// TIA Portal project "SVO_Lib" (V14)

(* hardware
DEVICE "S7300/ET200M station_1"  S7-300 station
   slot 0: "Rail_0"  Rail  6ES7 390-1***0-0AA0
   slot 2: "PLC_300"  CPU 315-2 PN/DP  6ES7 315-2EH14-0AB0  V3.2
      slot 2: "PROFINET interface_1"  PN-IO
         slot 1: "Port_1"  Port
         slot 2: "Port_2"  Port
   slot 4: "DI 8x120/230VAC_1"  DI8 x 230VAC  6ES7 321-1FF01-0AA0
DEVICE "S7-1200 station_1"  S7-1200 Station
   slot 0: "Rack_0"  S7-1200 Rack  Rack  V1.0
   slot 1: "PLC_1200"  CPU 1217C DC/DC/DC  6ES7 217-1AG40-0XB0  V4.2
DEVICE "HMI_1"  TP900 Comfort
   slot 0: "TP900 Comfort"  TP900 Comfort  6AV2 124-0JC01-0AX0  14.0.1.0
   slot 1: "HMI_RT_1"  TP900 Comfort  6AV2 124-0JC01-0AX0  14.0.1.0
   slot 5: "HMI_1.IE_CP_1"  PROFINET Interface  14.0.1.0
      slot 1: "PROFINET Interface_1"  PROFINET Interface
         slot 1: "Port_1"  Port
         slot 2: "Port_2"  Port
   slot 7: "HMI_1.MPI/DP_CP_1"  MPI/DP Interface  14.0.1.0
*)

// ===== PLC "PLC_300"  CPU 315-2 PN/DP =====

VAR_GLOBAL   // PLC tag table "Default tag table"
   "Tag_3" AT %M1.5 : Bool;
   "Tag_4" AT %M2.0 : Bool;
   "Tag_5" AT %M2.1 : Bool;
   "Tag_6" AT %M2.2 : Bool;
   "Tag_7" AT %MW4 : Int;
   "i0.0" AT %I0.0 : Bool;
   "i0.1" AT %I0.1 : Bool;
   "i0.2" AT %I0.2 : Bool;
   "i0.3" AT %I0.3 : Bool;
   "i0.4" AT %I0.4 : Bool;
   "i0.5" AT %I0.5 : Bool;
   "i0.6" AT %I0.6 : Bool;
   "i0.7" AT %I0.7 : Bool;
   "Tag_1" AT %M3.0 : Bool;
   "Tag_2" AT %M2.5 : Bool;
   "Tag_8" AT %M2.7 : Bool;
   "Tag_9" AT %M2.6 : Bool;
   "Tag_10" AT %MW20 : Int;
   "Tag_11" AT %MW22 : Int;
   "Tag_12" AT %MW24 : Int;
   "Tag_13" AT %MB26 : Byte;
   "Tag_14" AT %MB27 : Byte;
   "Tag_15" AT %MB28 : Byte;
   "Tag_16" AT %MB29 : Byte;
   "Tag_17" AT %MB30 : Byte;
   "Tag_18" AT %MB31 : Byte;
   "Tag_19" AT %MB32 : Byte;
   "Tag_20" AT %MB33 : Byte;
END_VAR

VAR_GLOBAL CONSTANT   // PLC tag table "Default tag table"
   "T" : Bool := 1;
   "T2" : Bool := true;
END_VAR

VAR_GLOBAL   // PLC tag table "PLCTagsKernel"
   "Blink0_1s" AT %M10.0 : Bool;   // Frequency 10Гц
   "Blink0_2s" AT %M10.1 : Bool;   // Frequency 5Гц
   "Blink0_4s" AT %M10.2 : Bool;   // Frequency 2,5Гц
   "Blink0_5s" AT %M10.3 : Bool;   // Frequency 2Гц
   "Blink0_8s" AT %M10.4 : Bool;   // Frequency 1,25Гц
   "Blink1_0s" AT %M10.5 : Bool;   // Frequency 1Гц
   "Blink1_6s" AT %M10.6 : Bool;   // Frequency 0,625Гц
   "Blink2_0s" AT %M10.7 : Bool;   // Frequency 0,5Гц
   "False0" AT %M0.0 : Bool;   // Always 0 [No]
   "True1" AT %M0.1 : Bool;   // Always 1 [Yes]
   "PLC_Run" AT %M0.2 : Bool;   // PLC is run. [0:Stop, 1:Run]
   "COM_RST" AT %M0.3 : Bool;   // PLC was restart. [0:Stop or Run, 1:First cycle]
   "Dummy" AT %M0.6 : Bool;   // Do nothing.
   "Temp" AT %M0.7 : Bool;   // Will be change.[Mark from programmer]
   "PLC_Runing" AT %M0.4 : Bool;
END_VAR

TYPE "udtDI"
   STRUCT
      ibInput : Bool := false;   // Input signal from DI
      ibSimulationOn : Bool := false;   // When simulation is on Out = 1 [0:Off, 1:On]
      ibSensorsBipolar : Bool := false;   // [0:Unopolar,1:Bipolar]
      ibEnUseDelay : Bool := true;   // Enable use delay [0:Disable,1:Enable]
      iiOnDelaySP : Int := 1;   // Set point on delay [s]
      iiOffDelaySP : Int := 1;   // Set point off delay [s]
      ibBlink1s : Bool := false;   // A flickering signal with a frequency of 1s.
      obOut : Bool := false;   // Output signal to user program.
      niCountDelayOn : Int := 0;   // Time passed after on. Out memory for save.
      niCountDelayOff : Int := 0;   // Time passed after off. Out memory for save.
      nwStatusWord : Word := 16#0;   // Status word.
   END_STRUCT;
END_TYPE

DATA_BLOCK "diMunitorByDI"   // DB1
{ S7_Optimized_Access := 'FALSE' }
VERSION : 0.1
// stored: InstanceOfName fMonitorByDI
"fMonitorByDI"
BEGIN
END_DATA_BLOCK

DATA_BLOCK "O"   // DB2
{ S7_Optimized_Access := 'FALSE' }
VERSION : 0.1
   VAR
      DI : Array[0..100] of "udtDI";
   END_VAR
BEGIN
END_DATA_BLOCK

DATA_BLOCK "diMunitorByDI2"   // DB3
{ S7_Optimized_Access := 'FALSE' }
VERSION : 0.1
// stored: InstanceOfName fMonitorByDI
"fMonitorByDI"
BEGIN
END_DATA_BLOCK

DATA_BLOCK "fConvertWordToBits_DB"   // DB4
{ S7_Optimized_Access := 'FALSE' }
VERSION : 0.1
// stored: InstanceOfName fConvertWordToBits
"fConvertWordToBits"
BEGIN
END_DATA_BLOCK

DATA_BLOCK "fConvertByteToBits_DB"   // DB6
{ S7_Optimized_Access := 'FALSE' }
VERSION : 0.1
// stored: InstanceOfName fConvertByteToBits
"fConvertByteToBits"
BEGIN
END_DATA_BLOCK

FUNCTION_BLOCK "fConvertWordToBits"   // FB1, SCL
{ S7_Optimized_Access := 'FALSE' }
VERSION : 0.1
   VAR_INPUT
      iWord : Word := 16#0000;
   END_VAR
   VAR_OUTPUT
      oBit00 : Bool;
      oBit01 : Bool;
      oBit02 : Bool;
      oBit03 : Bool;
      oBit04 : Bool;
      oBit05 : Bool;
      oBit06 : Bool;
      oBit07 : Bool;
      oBit08 : Bool;
      oBit09 : Bool;
      oBit10 : Bool;
      oBit11 : Bool;
      oBit12 : Bool;
      oBit13 : Bool;
      oBit14 : Bool;
      oBit15 : Bool;
   END_VAR
   VAR_TEMP
      tWord : Word;
      arrayATtWord AT tWord : Array[0..15] of Bool;
   END_VAR
BEGIN
   (*
   Autor: Svinarenko V.O.
   Version : 1.0
   Notes:
   This function can unpack input word to bool.
   *)

   #tWord := #iWord;

   #oBit00 := #arrayATtWord[8];
   #oBit01 := #arrayATtWord[9];
   #oBit02 := #arrayATtWord[10];
   #oBit03 := #arrayATtWord[11];
   #oBit04 := #arrayATtWord[12];
   #oBit05 := #arrayATtWord[13];
   #oBit06 := #arrayATtWord[14];
   #oBit07 := #arrayATtWord[15];
   #oBit08 := #arrayATtWord[0];
   #oBit09 := #arrayATtWord[1];
   #oBit10 := #arrayATtWord[2];
   #oBit11 := #arrayATtWord[3];
   #oBit12 := #arrayATtWord[4];
   #oBit13 := #arrayATtWord[5];
   #oBit14 := #arrayATtWord[6];
   #oBit15 := #arrayATtWord[7];
END_FUNCTION_BLOCK

FUNCTION_BLOCK "fConvertBitsToWord"   // FB2, SCL
{ S7_Optimized_Access := 'FALSE' }
VERSION : 0.1
   VAR_INPUT
      iBit00 : Bool := FALSE;
      iBit01 : Bool := FALSE;
      iBit02 : Bool := FALSE;
      iBit03 : Bool := FALSE;
      iBit04 : Bool := FALSE;
      iBit05 : Bool := FALSE;
      iBit06 : Bool := FALSE;
      iBit07 : Bool := FALSE;
      iBit08 : Bool := FALSE;
      iBit09 : Bool := FALSE;
      iBit10 : Bool := FALSE;
      iBit11 : Bool := FALSE;
      iBit12 : Bool := FALSE;
      iBit13 : Bool := FALSE;
      iBit14 : Bool := FALSE;
      iBit15 : Bool := FALSE;
   END_VAR
   VAR_OUTPUT
      oWord : Word;
   END_VAR
   VAR_TEMP
      tWord : Word;
      arrayTWord AT tWord : Array[0..15] of Bool;
   END_VAR
BEGIN
   (*
   Autor: Svinarenko V.O.
   Version : 1.0
   Notes:
   This function can pack input bool to word.
   *)    
   #arrayTWord[0] := #iBit08;
   #arrayTWord[1] := #iBit09;
   #arrayTWord[2] := #iBit10;
   #arrayTWord[3] := #iBit11;
   #arrayTWord[4] := #iBit12;
   #arrayTWord[5] := #iBit13;
   #arrayTWord[6] := #iBit14;
   #arrayTWord[7] := #iBit15;
   #arrayTWord[8] := #iBit00;
   #arrayTWord[9] := #iBit01;
   #arrayTWord[10] := #iBit02;
   #arrayTWord[11] := #iBit03;
   #arrayTWord[12] := #iBit04;
   #arrayTWord[13] := #iBit05;
   #arrayTWord[14] := #iBit06;
   #arrayTWord[15] := #iBit07;

   #oWord := #tWord;
END_FUNCTION_BLOCK

FUNCTION_BLOCK "fMonitorByAI"   // FB3, SCL
{ S7_Optimized_Access := 'FALSE' }
VERSION : 0.1
   VAR_INPUT
      iiSCALE_IN : Int;   // Input value from analog input (PIW).
      iiSCALE_HI_Lim : Real := 100.0;   // High limit.
      iiSCALE_LO_Lim : Real := 0.0;   // Low limit.
      irLimHH : Real := 95.0;   // High alarm limit.
      irLimH : Real := 90.0;   // High warning limit.
      irHTL : Real := 60.0;   // High tolerant limit.
      irSP : Real := 50.0;   // Set point
      irLTL : Real := 40.0;   // Low tolerant limit.
      irLimL : Real := 10.0;   // Low warning limit.
      irLimLL : Real := 5.0;   // Low alarm limit.
      ibSimulationOn : Bool;
      ibBipolar : Bool := false;   // 0:unipolar, 1:Bipolar
      ibDoUseHiLim : Bool := true;   // 0: Do not use; 1: Use.
      ibDoUseLoLim : Bool := true;   // 0: Do not use; 1: Use.
   END_VAR
BEGIN


   // "fAICheckInputParam"(irLimHH:=#irLimHH,
   //                      irLimH:=#irLimH,
   //                      irLimL:=#irLimL,
   //                      irLimLL:=#irLimLL,
   //                      obParamOk=>_bool_out_);

   // "fAIScale"(ibBipolar:=#ibBipolar,
   //            iiSCALE_IN:=#iiSCALE_IN,
   //            iiSCALE_HI_Lim:=#iiSCALE_HI_Lim,
   //            iiSCALE_LO_Lim:=#iiSCALE_LO_Lim,
   //            orPV=>_real_out_);


   // "fAICheckLim"(irPV:=_real_in_,
   //               irLimHH:=#irLimHH,
   //               irLimH:=#irLimH,
   //               irHTL:=#irHTL,
   //               irLTL:=#irLTL,
   //               irLimL:=#irLimL,
   //               irLimLL:=#irLimLL,
   //               ibDoUseHiLim:=#ibDoUseHiLim,
   //               ibDoUseLoLim:=#ibDoUseLoLim,
   //               obFlt=>_bool_out_,
   //               obWrn=>_bool_out_,
   //               obTolerant=>_bool_out_,
   //               obFltHH=>_bool_out_,
   //               obWrnH=>_bool_out_,
   //               obWrnL=>_bool_out_,
   //               obFltLL=>_bool_out_);

   (*
   Status 
   0 Bag - Red
   1 HH - Red
   2 H - Yelow
   3 N - Gray
   4 T - Green
   5 N - Gray
   6 L - Yelow
   7 LL - Red
   *)
END_FUNCTION_BLOCK

FUNCTION_BLOCK "fValve"   // FB4, SCL
{ S7_Optimized_Access := 'FALSE' }
VERSION : 0.1
   VAR_INPUT
      ibAutoMode : Bool;
      ibManMode : Bool;
      ibAutoGoOpen : Array[0..7] of Bool;
      ibManGoOpenFromHMI : Bool;
      ibManGoOpenFromBtnFlipFlop : Bool;
      ibManGoOpenFromSwich : Bool;
      ibManGoOpenFromBtnStart : Bool;
      ibManGoOpenFromBtnStop : Bool;
      ibLook : Bool;
      ibValveIsOpen : Bool;
      ibValveIsClose : Bool;
      iiTime : Int;
   END_VAR
BEGIN
END_FUNCTION_BLOCK

FUNCTION_BLOCK "fConvertByteToBits"   // FB5, SCL
{ S7_Optimized_Access := 'FALSE' }
VERSION : 0.1
   VAR_INPUT
      iByte : Byte := 16#0000;
   END_VAR
   VAR_OUTPUT
      oBit00 : Bool;
      oBit01 : Bool;
      oBit02 : Bool;
      oBit03 : Bool;
      oBit04 : Bool;
      oBit05 : Bool;
      oBit06 : Bool;
      oBit07 : Bool;
   END_VAR
   VAR_TEMP
      tByte : Byte;
      arrayATtByte AT tByte : Array[0..7] of Bool;
   END_VAR
BEGIN
   (*
   Autor: Svinarenko V.O.
   Version : 1.0
   Notes:
   This function can unpack input byte to bool.
   *)

   #tByte := #iByte;

   #oBit00 := #arrayATtByte[0];
   #oBit01 := #arrayATtByte[1];
   #oBit02 := #arrayATtByte[2];
   #oBit03 := #arrayATtByte[3];
   #oBit04 := #arrayATtByte[4];
   #oBit05 := #arrayATtByte[5];
   #oBit06 := #arrayATtByte[6];
   #oBit07 := #arrayATtByte[7];
END_FUNCTION_BLOCK

FUNCTION_BLOCK "fMonitorByDI"   // FB50, SCL
TITLE = fMunitorByDI
{ S7_Optimized_Access := 'FALSE' }
AUTHOR : SVO
FAMILY : Munitor
VERSION : 1.2
   VAR_INPUT
      ibInput : Bool;   // Input signal from DI
      ibSimulationOn : Bool;   // When simulation is on we monitor input ibSimulationIn [0:Off, 1:On]
      ibSimulationIn : Bool;   // When simulation is on Out = 1 [0:Off, 1:On]
      ibSensorsBipolar : Bool;   // [0:Unopolar,1:Bipolar]
      ibEnUseDelay : Bool;   // Enable use delay [0:Disable,1:Enable]
      iiOnDelaySP : Int := 1;   // Set point on delay [s]
      iiOffDelaySP : Int := 1;   // Set point off delay [s]
      ibBlink1s : Bool;   // A flickering signal with a frequency of 1s.
   END_VAR
   VAR_OUTPUT
      obOut : Bool;   // Output signal to user program.
   END_VAR
   VAR_IN_OUT
      niCountDelayOn : Int;   // Time passed after on. Out memory for save.
      niCountDelayOff : Int;   // Time passed after off. Out memory for save.
      nwStatusWord : Word;   // Status word.
   END_VAR
   VAR
      sfWordToBits : "fConvertWordToBits";   // Convert word to bits.
      sfBitsToWord : "fConvertBitsToWord";   // Convert bits to word.
   END_VAR
   VAR_TEMP
      tb_swb0_Input : Bool;
      tb_swb1_Out : Bool;
      tb_swb2_TimeOnFinish : Bool;
      tb_swb3_TimeOnFrontBlink : Bool;
      tb_swb4_TimeOffFinish : Bool;
      tb_swb5_TimeOffFrontBlink : Bool;
      tb_swb6 : Bool;
      tb_swb7 : Bool;
      tb_swb8_AlarmParamIsNotCorect : Bool;
      tb_swb9 : Bool;
      tb_swb10 : Bool;
      tb_swb11 : Bool;
      tb_swb12 : Bool;
      tb_swb13 : Bool;
      tb_swb14 : Bool;
      tb_swb15 : Bool;
      tiCorectTimeOnDelaySP : Int;
      tiCorectTimeOffDelaySP : Int;
   END_VAR
BEGIN
   (*
   Autor: Svinarenko V.O.
   Version : 1.1
   Note:
   This function monitor by digital input, it can:
   *Inver input signal (param ibSensorIsBipolar);
   *Create delay (ibEnUseDelay);
   **On delay (paramiiOnDelaySP);
   **Off delay (paramiiOffDelaySP);
   *Form status word.

   Releases : v1.1 by 2018 01 23 
   Timer IEC_TON has been replaced by fCount.

   Releases : v1.2 by 2018 01 25
   The CheckInputParam has been added.

   Releases : v1.3 by 2018 05 23
   Add input ibSimulationIn.
   *)

   REGION rCheckInputParam
       //Setpoint for timer can't be lower than 0.
       //If Delay is on than all setpoint can't be equal 0. It is equal Delay = Off. 
       IF (#ibEnUseDelay AND (#iiOnDelaySP = 0) AND (#iiOffDelaySP = 0)) OR (#iiOnDelaySP < 0) OR (#iiOffDelaySP < 0) THEN
           #tb_swb8_AlarmParamIsNotCorect := true;//We creat alarm for OP.
           #tiCorectTimeOnDelaySP := 1;
           #tiCorectTimeOffDelaySP := 1;
       ELSE
           #tb_swb8_AlarmParamIsNotCorect := false;
           #tiCorectTimeOnDelaySP := #iiOnDelaySP;
           #tiCorectTimeOffDelaySP := #iiOffDelaySP;
       END_IF;
   END_REGION


   REGION rUnpackStatusWord
       //This function unpack status word to bit. All data must be saved outside function.
       //When data saved outside functon, we can use this function in loop for DI masif.
       #sfWordToBits(iWord := #nwStatusWord,
                     oBit00 => #tb_swb0_Input,
                     oBit01 => #tb_swb1_Out,
                     oBit02 => #tb_swb2_TimeOnFinish,
                     oBit03 => #tb_swb3_TimeOnFrontBlink,
                     oBit04 => #tb_swb4_TimeOffFinish,
                     oBit05 => #tb_swb5_TimeOffFrontBlink,
                     oBit06 => #tb_swb6,
                     oBit07 => #tb_swb7,
                     oBit08 => #tb_swb8_AlarmParamIsNotCorect,
                     oBit09 => #tb_swb9,
                     oBit10 => #tb_swb10,
                     oBit11 => #tb_swb11,
                     oBit12 => #tb_swb12,
                     oBit13 => #tb_swb13,
                     oBit14 => #tb_swb14,
                     oBit15 => #tb_swb15);
   END_REGION
   REGION rBipolar
       IF #ibSensorsBipolar THEN
           #tb_swb0_Input := NOT #ibInput;
       ELSE
           #tb_swb0_Input := #ibInput;
       END_IF;
   END_REGION

   REGION rDelay
       IF #ibEnUseDelay THEN
           //When the Delay is on, Out will swich after delay 
           //Delay on Out
           "fCount"(ibStartTimer := #tb_swb0_Input,
                    ibBlink1s := #ibBlink1s,
                    iiTimeSP := #tiCorectTimeOnDelaySP,
                    obFinish => #tb_swb2_TimeOnFinish,
                    niCount := #niCountDelayOn,
                    nbFrontBlink := #tb_swb3_TimeOnFrontBlink);
           //Delay off Out
           "fCount"(ibStartTimer := NOT #tb_swb0_Input,
                    ibBlink1s := #ibBlink1s,
                    iiTimeSP := #tiCorectTimeOffDelaySP,
                    obFinish => #tb_swb4_TimeOffFinish,
                    niCount := #niCountDelayOff,
                    nbFrontBlink := #tb_swb5_TimeOffFrontBlink);
       ELSE
           #tb_swb2_TimeOnFinish := false;
           #tb_swb4_TimeOffFinish := false;
       END_IF;
   END_REGION

   REGION rOut
       IF NOT #ibSimulationOn THEN //When simulation is on Out  = ibSimulationI
           IF #ibEnUseDelay THEN //When the Delay is on, the Out turn on after the delay. 
               IF #tb_swb2_TimeOnFinish THEN
                   #tb_swb1_Out := TRUE;
               END_IF;
               IF #tb_swb4_TimeOffFinish THEN
                   #tb_swb1_Out := False;
               END_IF;
           ELSE //When the Delay is off, input signal go to output.
               #tb_swb1_Out := #tb_swb0_Input;
           END_IF;
       ELSE //When simulation is on Out  = 1
           #tb_swb1_Out := #ibSimulationIn;
       END_IF;
       #obOut := #tb_swb1_Out;
   END_REGION

   REGION rPackStatusWord
       //This function pack bit to status word. All data must be saved outside function.
       //When data saved outside functon, we can use this function in loop for DI masif.
       #sfBitsToWord(iBit00 := #tb_swb0_Input,
                     iBit01 := #tb_swb1_Out,
                     iBit02 := #tb_swb2_TimeOnFinish,
                     iBit03 := #tb_swb3_TimeOnFrontBlink,
                     iBit04 := #tb_swb4_TimeOffFinish,
                     iBit05 := #tb_swb5_TimeOffFrontBlink,
                     iBit06 := #tb_swb6,
                     iBit07 := #tb_swb7,
                     iBit08 := #tb_swb8_AlarmParamIsNotCorect,
                     iBit09 := #tb_swb9,
                     iBit10 := #tb_swb10,
                     iBit11 := #tb_swb11,
                     iBit12 := #tb_swb12,
                     iBit13 := #tb_swb13,
                     iBit14 := #tb_swb14,
                     iBit15 := #tb_swb15,
                     oWord => #nwStatusWord);
   END_REGION
END_FUNCTION_BLOCK

FUNCTION "fCount" : Void   // FC1, SCL
{ S7_Optimized_Access := 'FALSE' }
VERSION : 0.1
   VAR_INPUT
      ibStartTimer : Bool;   // Start time countdown [0:Stop, 1:Start]
      ibBlink1s : Bool;   // Blink with frequency 1s [Mx.5]
      iiTimeSP : Int;   // Set point time. [s]
   END_VAR
   VAR_OUTPUT
      obFinish : Bool;   // The countdown is finish.
   END_VAR
   VAR_IN_OUT
      niCount : Int;   // Passed time. [s]
      nbFrontBlink : Bool;   // Front positive.
   END_VAR
BEGIN
   IF #ibStartTimer THEN
       IF #ibBlink1s AND NOT #nbFrontBlink THEN
           #niCount := #niCount + 1;
           #nbFrontBlink := true;
       END_IF;
       IF NOT #ibBlink1s THEN
           #nbFrontBlink := false;
       END_IF;
   ELSE
       #niCount := 0;
   END_IF;

   IF #niCount >= #iiTimeSP THEN
       #obFinish := TRUE;
       #niCount := #iiTimeSP;
   ELSE
       #obFinish := FALSE;
   END_IF;
END_FUNCTION

FUNCTION "call" : Void   // FC2, SCL
{ S7_Optimized_Access := 'FALSE' }
VERSION : 0.1
   VAR_TEMP
      i : Int;
   END_VAR
BEGIN
   "O".DI[0].ibInput := "i0.0";
   "O".DI[1].ibInput := "i0.1";
   "O".DI[2].ibInput := "i0.2";
   "O".DI[3].ibInput := "i0.3";
   "O".DI[4].ibInput := "i0.4";
   "O".DI[5].ibInput := "i0.5";
   "O".DI[6].ibInput := "i0.6";
   "O".DI[7].ibInput := "i0.7";


   FOR #i := 0 TO 7 DO
       // "diMunitorByDI2"(ibInput := "O".DI[#i].ibInput,
       //                  ibSensorIsBipolar := "O".DI[#i].ibSensorIsBipolar,
       //                  ibEnUseDelay := "O".DI[#i].ibEnUseDelay,
       //                  iiOnDelaySP := "O".DI[#i].iiOnDelaySP,
       //                  iiOffDelaySP := "O".DI[#i].iiOffDelaySP,
       //                  ibBlink1s := "Tag_3",
       //                  obOut => "O".DI[#i].obOut,
       //                  niCountDelayOn := "O".DI[#i].niCountDelayOn,
       //                  niCountDelayOff := "O".DI[#i].niCountDelayOff,
       //                  nwStatusWord := "O".DI[#i].nwStatusWord);
       ;
   END_FOR;
END_FUNCTION

FUNCTION "fAIScale" : Void   // FC3, SCL
{ S7_Optimized_Access := 'FALSE' }
VERSION : 0.1
   VAR_INPUT
      ibBipolar : Bool;   // 0:unipolar, 1:Bipolar
      iiSCALE_IN : Int;   // Input value from analog input (PIW).
      iiSCALE_HI_Lim : Real;   // High limit.
      iiSCALE_LO_Lim : Real;   // Low limit.
   END_VAR
   VAR_OUTPUT
      orPV : Real;   // Output value in physics units.
   END_VAR
   VAR_TEMP
      tiNormaleMin : Int;   // Min
      trNormaleOut : Real;   // Normalized value from 0.0 to 1.0
   END_VAR
   VAR CONSTANT
      ciNormaleMax : Int := 27648;   // Max
   END_VAR
BEGIN
   (*
   Autor: Svinarenko V.O.
   Version : 1.0
   Note:
   This function convert input value from PIW to output value in  physics units.
   *)
   IF #ibBipolar THEN
       #tiNormaleMin := -27648;
   ELSE
       #tiNormaleMin := 0;
   END_IF;
   #trNormaleOut := (#iiSCALE_IN - #tiNormaleMin) / (#ciNormaleMax - #tiNormaleMin); //Convert input value from PIW to normale value from 0.0 to 1.0
   #orPV := (#trNormaleOut * (#iiSCALE_HI_Lim - #iiSCALE_LO_Lim)) + #iiSCALE_LO_Lim; //Normale value convert to physical units
END_FUNCTION

FUNCTION "fAICheckInputParam" : Void   // FC4, SCL
{ S7_Optimized_Access := 'FALSE' }
VERSION : 0.1
   VAR_INPUT
      irLimHH : Real;   // High alarm limit.
      irLimH : Real;   // High warning limit.
      irLimL : Real;   // Low warning limit.
      irLimLL : Real;   // Low alarm limit.
   END_VAR
   VAR_OUTPUT
      obParamOk : Bool;   // 0: Input parameters are corect. 1: Input parameters are not corect
   END_VAR
BEGIN
   (*
   Autor: Svinarenko V.O.
   Version : 1.0
   Note:
   This function check input parameters.
   *)
   #obParamOk := true;
   IF #irLimLL > #irLimL THEN
       #obParamOk := false;
   END_IF;
   IF #irLimL > #irLimH THEN
       #obParamOk := false;
   END_IF;
   IF #irLimH > #irLimHH THEN
       #obParamOk := false;
   END_IF;
END_FUNCTION

FUNCTION "fAICheckLim" : Void   // FC5, SCL
{ S7_Optimized_Access := 'FALSE' }
VERSION : 0.1
   VAR_INPUT
      irPV : Real;   // Value in physics units.
      irLimHH : Real;   // High alarm limit.
      irLimH : Real;   // High warning limit.
      irHTL : Real;   // High tolerant limit.
      irLTL : Real;   // Low tolerant limit.
      irLimL : Real;   // Low warning limit.
      irLimLL : Real;   // Low alarm limit.
      ibDoUseHiLim : Bool;   // 0: Do not use; 1: Use.
      ibDoUseLoLim : Bool;   // 0: Do not use; 1: Use.
   END_VAR
   VAR_OUTPUT
      obFlt : Bool;   // The current value has crossed alarm limit.
      obWrn : Bool;   // The current value has crossed warning limit.
      obTolerant : Bool;   // The current value is tolerant.
      obFltHH : Bool;   // The current value is over then the upper alarm limit.
      obWrnH : Bool;   // The current value is over then the upper warning limit.
      obWrnL : Bool;   // The current value is lower then the low warning limit.
      obFltLL : Bool;   // The current value is lower then the low alarm limit.
   END_VAR
BEGIN
   (*
   Autor: Svinarenko V.O.
   Version : 1.0
   Note:
   This function check input value and create alarm or warning.
   *)
   #obFlt := #irPV > #irLimHH AND #ibDoUseHiLim OR #irPV < #irLimLL AND #ibDoUseLoLim;
   #obFltHH := (#irPV > #irLimHH) AND #ibDoUseHiLim;
   #obFltLL := #irPV < #irLimLL AND #ibDoUseLoLim;
   #obWrn := #irPV > #irLimH AND #ibDoUseHiLim OR #irPV < #irLimL AND #ibDoUseLoLim;
   #obWrnH := #irPV > #irLimH AND #ibDoUseHiLim;
   #obWrnL := #irPV < #irLimL AND #ibDoUseLoLim;

   #obTolerant := (#irPV > #irLTL) AND (#irPV < #irHTL);
END_FUNCTION

FUNCTION "FCInitialization" : Void   // FC6, SCL
{ S7_Optimized_Access := 'FALSE' }
VERSION : 0.1
BEGIN
   (*
   Autor: Svinarenko V.O.
   Version : 1.0
   Note:
   This function initializating CONSTANTS.

   Releases : v1.0 by 2018 05 23
   Function was creating.
   *)
   "False0" := FALSE;
   "True1" := TRUE;
END_FUNCTION

FUNCTION "FC_CompleteRestart" : Void   // FC7, SCL
{ S7_Optimized_Access := 'FALSE' }
VERSION : 0.1
   VAR_INPUT
      ibComRst : Bool;
   END_VAR
BEGIN
   "COM_RST" := #ibComRst;
END_FUNCTION

ORGANIZATION_BLOCK "MAIN"   // OB1, LAD
TITLE = "Main Program Sweep (Cycle)"
{ S7_Optimized_Access := 'FALSE' }
VERSION : 0.1
   VAR_TEMP
      OB1_EV_CLASS : Byte;   // Bits 0-3 = 1 (Coming event), Bits 4-7 = 1 (Event class 1)
      OB1_SCAN_1 : Byte;   // 1 (Cold restart scan 1 of OB 1), 3 (Scan 2-n of OB 1)
      OB1_PRIORITY : Byte;   // Priority of OB Execution
      OB1_OB_NUMBR : Byte;   // 1 (Organization block 1, OB1)
      OB1_RESERVED_1 : Byte;   // Reserved for system
      OB1_RESERVED_2 : Byte;   // Reserved for system
      OB1_PREV_CYCLE : Int;   // Cycle time of previous OB1 scan (milliseconds)
      OB1_MIN_CYCLE : Int;   // Minimum cycle time of OB1 (milliseconds)
      OB1_MAX_CYCLE : Int;   // Maximum cycle time of OB1 (milliseconds)
      OB1_DATE_TIME : Date_And_Time;   // Date and time OB1 started
   END_VAR
   VAR_TEMP   // added for the SCL form of the ladder/FBD networks
      _w1 : Bool;
   END_VAR
BEGIN

REGION Network 1
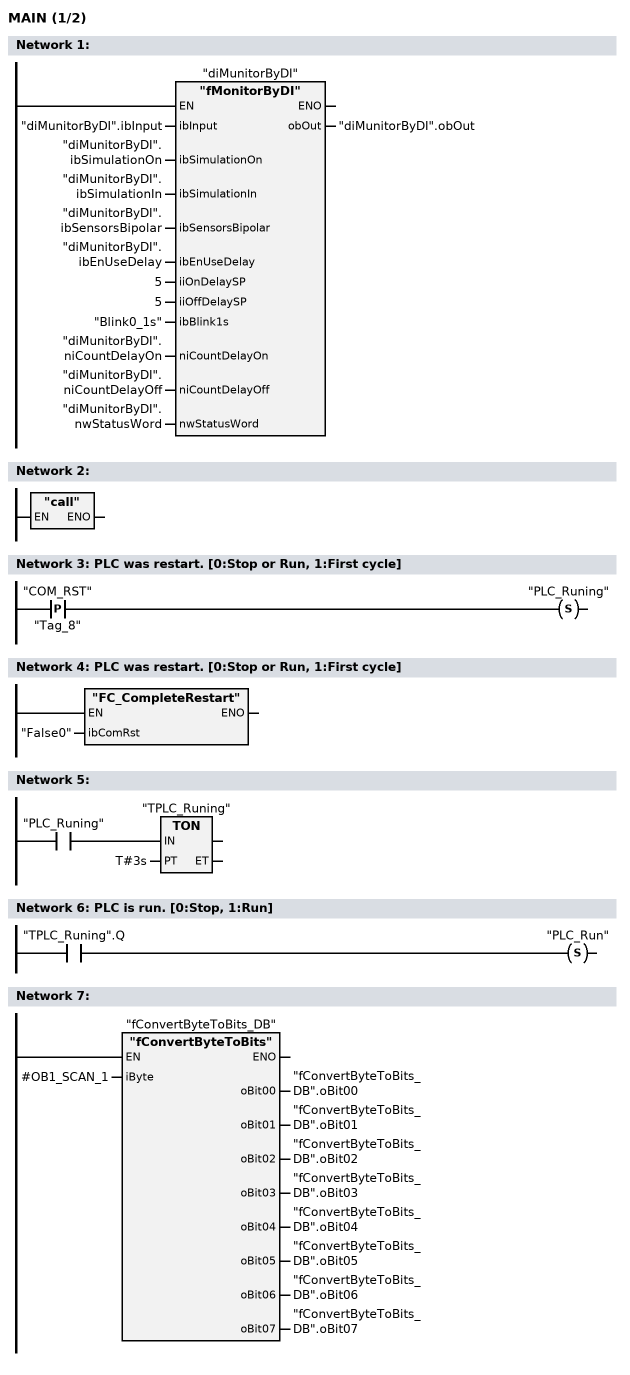
   RUNG wire#powerrail
      "diMunitorByDI"(ibInput := "diMunitorByDI".ibInput, ibSimulationOn := "diMunitorByDI".ibSimulationOn, ibSimulationIn := "diMunitorByDI".ibSimulationIn, ibSensorsBipolar := "diMunitorByDI".ibSensorsBipolar, ibEnUseDelay := "diMunitorByDI".ibEnUseDelay, iiOnDelaySP := 5, iiOffDelaySP := 5, ibBlink1s := "Blink0_1s", niCountDelayOn := "diMunitorByDI".niCountDelayOn, niCountDelayOff := "diMunitorByDI".niCountDelayOff, nwStatusWord := "diMunitorByDI".nwStatusWord, obOut => "diMunitorByDI".obOut)
   END_RUNG
   // the same network as SCL:
   "diMunitorByDI"(ibInput := "diMunitorByDI".ibInput,   // "fMonitorByDI"
                   ibSimulationOn := "diMunitorByDI".ibSimulationOn,
                   ibSimulationIn := "diMunitorByDI".ibSimulationIn,
                   ibSensorsBipolar := "diMunitorByDI".ibSensorsBipolar,
                   ibEnUseDelay := "diMunitorByDI".ibEnUseDelay,
                   iiOnDelaySP := 5,
                   iiOffDelaySP := 5,
                   ibBlink1s := "Blink0_1s",
                   niCountDelayOn := "diMunitorByDI".niCountDelayOn,
                   niCountDelayOff := "diMunitorByDI".niCountDelayOff,
                   nwStatusWord := "diMunitorByDI".nwStatusWord,
                   obOut => "diMunitorByDI".obOut);
END_REGION

REGION Network 2
   RUNG wire#powerrail
      "call"()
   END_RUNG
   // the same network as SCL:
   "call"();
END_REGION

REGION Network 3: PLC was restart. [0:Stop or Run, 1:First cycle]
   RUNG wire#powerrail
      P_Contact(operand := "COM_RST", bit := "Tag_8")
      S_Coil( "PLC_Runing" )
   END_RUNG
   // the same network as SCL:
   #_w1 := "COM_RST" AND NOT "Tag_8";   // rising edge of "COM_RST"
   "Tag_8" := "COM_RST";
   IF #_w1 THEN "PLC_Runing" := TRUE; END_IF;
END_REGION

REGION Network 4: PLC was restart. [0:Stop or Run, 1:First cycle]
   RUNG wire#powerrail
      "FC_CompleteRestart"(ibComRst := "False0")
   END_RUNG
   // the same network as SCL:
   "FC_CompleteRestart"(ibComRst := "False0");
END_REGION

REGION Network 5
   "TPLC_Runing".TON(IN := "PLC_Runing", PT := T#3s);
END_REGION

REGION Network 6: PLC is run. [0:Stop, 1:Run]
   RUNG wire#powerrail
      Contact( "TPLC_Runing".Q )
      S_Coil( "PLC_Run" )
   END_RUNG
   // the same network as SCL:
   IF "TPLC_Runing".Q THEN "PLC_Run" := TRUE; END_IF;
END_REGION

REGION Network 7
   RUNG wire#powerrail
      "fConvertByteToBits_DB"(iByte := #OB1_SCAN_1, oBit00 => "fConvertByteToBits_DB".oBit00, oBit01 => "fConvertByteToBits_DB".oBit01, oBit02 => "fConvertByteToBits_DB".oBit02, oBit03 => "fConvertByteToBits_DB".oBit03, oBit04 => "fConvertByteToBits_DB".oBit04, oBit05 => "fConvertByteToBits_DB".oBit05, oBit06 => "fConvertByteToBits_DB".oBit06, oBit07 => "fConvertByteToBits_DB".oBit07)
   END_RUNG
   // the same network as SCL:
   "fConvertByteToBits_DB"(iByte := #OB1_SCAN_1,   // "fConvertByteToBits"
                           oBit00 => "fConvertByteToBits_DB".oBit00,
                           oBit01 => "fConvertByteToBits_DB".oBit01,
                           oBit02 => "fConvertByteToBits_DB".oBit02,
                           oBit03 => "fConvertByteToBits_DB".oBit03,
                           oBit04 => "fConvertByteToBits_DB".oBit04,
                           oBit05 => "fConvertByteToBits_DB".oBit05,
                           oBit06 => "fConvertByteToBits_DB".oBit06,
                           oBit07 => "fConvertByteToBits_DB".oBit07);
END_REGION

REGION Network 8
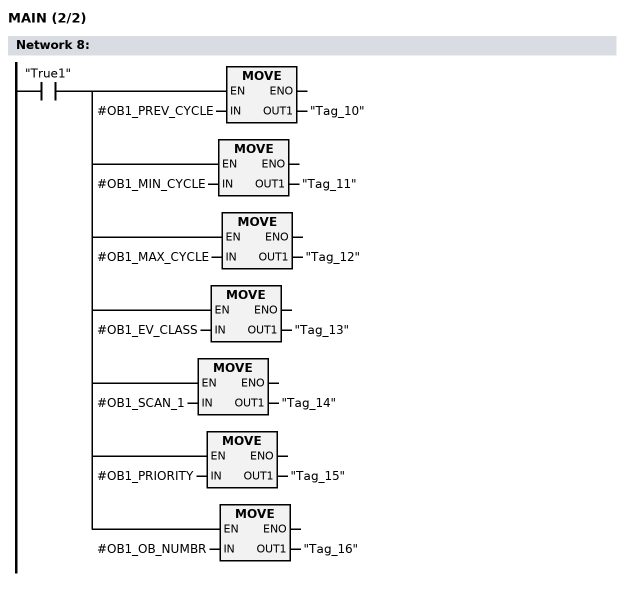
   RUNG wire#powerrail
      Contact( "True1" )
      wire#w1
      { S7_GenerateENO := "TRUE" } Move(in := #OB1_PREV_CYCLE, out1 => "Tag_10")
   END_RUNG
   RUNG wire#w1
      { S7_GenerateENO := "TRUE" } Move(in := #OB1_MIN_CYCLE, out1 => "Tag_11")
   END_RUNG
   RUNG wire#w1
      { S7_GenerateENO := "TRUE" } Move(in := #OB1_MAX_CYCLE, out1 => "Tag_12")
   END_RUNG
   RUNG wire#w1
      { S7_GenerateENO := "TRUE" } Move(in := #OB1_EV_CLASS, out1 => "Tag_13")
   END_RUNG
   RUNG wire#w1
      { S7_GenerateENO := "TRUE" } Move(in := #OB1_SCAN_1, out1 => "Tag_14")
   END_RUNG
   RUNG wire#w1
      { S7_GenerateENO := "TRUE" } Move(in := #OB1_PRIORITY, out1 => "Tag_15")
   END_RUNG
   RUNG wire#w1
      { S7_GenerateENO := "TRUE" } Move(in := #OB1_OB_NUMBR, out1 => "Tag_16")
   END_RUNG
   // the same network as SCL:
   IF "True1" THEN
       "Tag_10" := #OB1_PREV_CYCLE;
       "Tag_11" := #OB1_MIN_CYCLE;
       "Tag_12" := #OB1_MAX_CYCLE;
       "Tag_13" := #OB1_EV_CLASS;
       "Tag_14" := #OB1_SCAN_1;
       "Tag_15" := #OB1_PRIORITY;
       "Tag_16" := #OB1_OB_NUMBR;
   END_IF;
END_REGION
END_ORGANIZATION_BLOCK

ORGANIZATION_BLOCK "CYC_INT_100MS"   // OB35, SCL
TITLE = "Cyclic Interrupt"
{ S7_Optimized_Access := 'FALSE' }
VERSION : 0.1
   VAR_TEMP
      OB35_EV_CLASS : Byte;   // Bits 0-3 = 1 (Coming event), Bits 4-7 = 1 (Event class 1)
      OB35_STRT_INF : Byte;   // 16#36 (OB 35 has started)
      OB35_PRIORITY : Byte;   // Priority of OB Execution
      OB35_OB_NUMBR : Byte;   // 35 (Organization block 35, OB35)
      OB35_RESERVED_1 : Byte;   // Reserved for system
      OB35_RESERVED_2 : Byte;   // Reserved for system
      OB35_PHASE_OFFSET : Word;   // Phase offset (msec)
      OB35_RESERVED_3 : Int;   // Reserved for system
      OB35_EXC_FREQ : Int;   // Frequency of execution (msec)
      OB35_DATE_TIME : Date_And_Time;   // Date and time OB35 started
   END_VAR
BEGIN
   "Tag_17" := #OB35_EV_CLASS;
   "Tag_18" := #OB35_STRT_INF;
   "Tag_19" := #OB35_PRIORITY;
   "Tag_20" := #OB35_OB_NUMBR;
END_ORGANIZATION_BLOCK

ORGANIZATION_BLOCK "COMPLETE_RESTART"   // OB100, SCL
TITLE = "Complete Restart"
{ S7_Optimized_Access := 'FALSE' }
VERSION : 0.1
   VAR_TEMP
      OB100_EV_CLASS : Byte;   // 16#13, Event class 1, Entering event state, Event logged in diagnostic buffer
      OB100_STRTUP : Byte;   // 16#81/82/83/84 Method of startup
      OB100_PRIORITY : Byte;   // Priority of OB Execution
      OB100_OB_NUMBR : Byte;   // 100 (Organization block 100, OB100)
      OB100_RESERVED_1 : Byte;   // Reserved for system
      OB100_RESERVED_2 : Byte;   // Reserved for system
      OB100_STOP : Word;   // Event that caused CPU to stop (16#4xxx)
      OB100_STRT_INFO : DWord;   // Information on how system started
      OB100_DATE_TIME : Date_And_Time;   // Date and time OB100 started
   END_VAR
BEGIN
   "FC_CompleteRestart"(True);

   "PLC_Run" := FALSE;
   "PLC_Runing" := false;
END_ORGANIZATION_BLOCK

// ===== PLC "PLC_1200"  CPU 1217C DC/DC/DC =====

FUNCTION_BLOCK "fWordToBits"   // FB1, SCL
{ S7_Optimized_Access := 'FALSE' }
VERSION : 0.1
   VAR_INPUT
      iWord : Word := 16#0000;
   END_VAR
   VAR_OUTPUT
      oBit00 : Bool;
      oBit01 : Bool;
      oBit02 : Bool;
      oBit03 : Bool;
      oBit04 : Bool;
      oBit05 : Bool;
      oBit06 : Bool;
      oBit07 : Bool;
      oBit08 : Bool;
      oBit09 : Bool;
      oBit10 : Bool;
      oBit11 : Bool;
      oBit12 : Bool;
      oBit13 : Bool;
      oBit14 : Bool;
      oBit15 : Bool;
   END_VAR
   VAR_TEMP
      tWord : Word;
      arrayATtWord AT tWord : Array[0..15] of Bool;
   END_VAR
BEGIN
   (*
   Autor: Svinarenko V.O.
   Version : 1.0
   Notes:
   This function can unpack input word to bool.
   *)

   #tWord := #iWord;

   #oBit00 := #arrayATtWord[8];
   #oBit01 := #arrayATtWord[9];
   #oBit02 := #arrayATtWord[10];
   #oBit03 := #arrayATtWord[11];
   #oBit04 := #arrayATtWord[12];
   #oBit05 := #arrayATtWord[13];
   #oBit06 := #arrayATtWord[14];
   #oBit07 := #arrayATtWord[15];
   #oBit08 := #arrayATtWord[0];
   #oBit09 := #arrayATtWord[1];
   #oBit10 := #arrayATtWord[2];
   #oBit11 := #arrayATtWord[3];
   #oBit12 := #arrayATtWord[4];
   #oBit13 := #arrayATtWord[5];
   #oBit14 := #arrayATtWord[6];
   #oBit15 := #arrayATtWord[7];
END_FUNCTION_BLOCK

FUNCTION_BLOCK "fBitsToWord"   // FB2, SCL
{ S7_Optimized_Access := 'FALSE' }
VERSION : 0.1
   VAR_INPUT
      iBit00 : Bool := FALSE;
      iBit01 : Bool := FALSE;
      iBit02 : Bool := FALSE;
      iBit03 : Bool := FALSE;
      iBit04 : Bool := FALSE;
      iBit05 : Bool := FALSE;
      iBit06 : Bool := FALSE;
      iBit07 : Bool := FALSE;
      iBit08 : Bool := FALSE;
      iBit09 : Bool := FALSE;
      iBit10 : Bool := FALSE;
      iBit11 : Bool := FALSE;
      iBit12 : Bool := FALSE;
      iBit13 : Bool := FALSE;
      iBit14 : Bool := FALSE;
      iBit15 : Bool := FALSE;
   END_VAR
   VAR_OUTPUT
      oWord : Word;
   END_VAR
   VAR_TEMP
      tWord : Word;
      arrayTWord AT tWord : Array[0..15] of Bool;
   END_VAR
BEGIN
   (*
   Autor: Svinarenko V.O.
   Version : 1.0
   Notes:
   This function can pack input bool to word.
   *)    
   #arrayTWord[0] := #iBit08;
   #arrayTWord[1] := #iBit09;
   #arrayTWord[2] := #iBit10;
   #arrayTWord[3] := #iBit11;
   #arrayTWord[4] := #iBit12;
   #arrayTWord[5] := #iBit13;
   #arrayTWord[6] := #iBit14;
   #arrayTWord[7] := #iBit15;
   #arrayTWord[8] := #iBit00;
   #arrayTWord[9] := #iBit01;
   #arrayTWord[10] := #iBit02;
   #arrayTWord[11] := #iBit03;
   #arrayTWord[12] := #iBit04;
   #arrayTWord[13] := #iBit05;
   #arrayTWord[14] := #iBit06;
   #arrayTWord[15] := #iBit07;

   #oWord := #tWord;
END_FUNCTION_BLOCK

ORGANIZATION_BLOCK "Main"   // OB1, LAD, ProgramCycle
TITLE = "Main Program Sweep (Cycle)"
{ S7_Optimized_Access := 'TRUE' }
VERSION : 0.1
   VAR_INPUT
      Initial_Call : Bool;   // Initial call of this OB
      Remanence : Bool;   // =True, if remanent data are available
   END_VAR
BEGIN
END_ORGANIZATION_BLOCK

(* ===== HMI "HMI_RT_1" =====
system functions are stored by id; their names below are inferred from use
connection "HMI_Connection_1": ETHERNET, SIMATIC S7 300/400 MPI

HMI tags "Default tag table"
   "Tag_ScreenNumber" : UInt, internal
   "diMunitorByDI_niCountDelayOff" : Int = PLC diMunitorByDI.niCountDelayOff AT %DB1.DBW12, 1 s
   "SW" : Word = PLC BitsToWord_DB.owWord AT %DB4.DBW2, 1 s

screen "Home" 800x420, template "Template_1"
   on GenerateScreen: SetTag("Tag_ScreenNumber", 1)
   TextField "HmiScreenItemData_4" at 80,167 size 640x22; Text 'Welcome to HMI_1 (TP900 Comfort)!'
   Button "HmiScreenItemData" at 36,36 size 159x47; TextOff 'Plan'; PictureOff "Navigates to Plan for TP900 Comfort 14.0.1.0"; PictureOn "Navigates to Plan for TP900 Comfort 14.0.1.0"
      on Release: ActivateScreen("Plan", 0)
   Button "HmiScreenItemData_1" at 36,95 size 159x47; TextOff 'Param'; PictureOff "Navigates to Param for TP900 Comfort 14.0.1.0"; PictureOn "Navigates to Param for TP900 Comfort 14.0.1.0"
      on Release: ActivateScreen("Param", 0)
   Button "HmiScreenItemData_2" at 36,154 size 159x47; TextOff 'Recipe'; PictureOff "Navigates to Recipe for TP900 Comfort 14.0.1.0"; PictureOn "Navigates to Recipe for TP900 Comfort 14.0.1.0"
      on Release: ActivateScreen("Recipe", 0)
   Button "HmiScreenItemData_3" at 36,213 size 159x47; TextOff 'Trend'; PictureOff "Navigates to Trend for TP900 Comfort 14.0.1.0"; PictureOn "Navigates to Trend for TP900 Comfort 14.0.1.0"
      on Release: ActivateScreen("Trend", 0)
   Button "HmiScreenItemData_5" at 36,272 size 159x47; TextOff 'System screens'; PictureOff "Navigates to System screens for TP900 Comfort 14.0.1.0"; PictureOn "Navigates to System screens for TP900 Comfort 14.0.1.0"
      on Release: ActivateScreen("System screens", 0)

Template "Template_1" 800x420
   Button "Exit" at 720,360 size 78x58; TextOff 'Exit'; PictureOff "ExitRuntime_TP900_Comfort_TR"; PictureOn "ExitRuntime_TP900_Comfort_TR"
      on Release: StopRuntime(0)
   Button "Log on" at 640,360 size 78x58; TextOff 'Log on'; PictureOff "Login_TP900_Comfort_TR"; PictureOn "Login_TP900_Comfort_TR"
      on Release: function_a2a04561()
   Button "Template_Button" at 560,360 size 78x58; TextOff 'Text'
   Button "Template_Button_1" at 480,360 size 78x58; TextOff 'Text'
   Button "Template_Button_2" at 400,360 size 78x58; TextOff 'Trend'
      on Press: ActivateScreen("Trend", 0)
   Button "Template_Button_3" at 321,360 size 78x58; TextOff 'Recipe'
      on Press: ActivateScreen("Recipe", 0)
   Button "Template_Button_4" at 241,360 size 78x58; TextOff 'Param'
      on Press: ActivateScreen("Param", 0)
   Button "Template_Button_5" at 161,360 size 78x58; TextOff 'Plan'
      on Press: ActivateScreen("Plan", 0)
   Button "Alarms" at 81,360 size 78x58; TextOff 'Alarms'; PictureOff "AlarmDisplay_TP900_Comfort_TR"; PictureOn "AlarmDisplay_TP900_Comfort_TR"
      on Release: function_ef3f5d25("Alarm window_Unacknowledged", -1)
   Button "Start screen" at 1,360 size 78x58; TextOff 'Start screen'; PictureOff "NavigateHome_TP900_Comfort_TR"; PictureOn "NavigateHome_TP900_Comfort_TR"
      on Release: ActivateScreen("Home", 0)

screen "Plan" 800x420, template "Template_1"
   on GenerateScreen: SetTag("Tag_ScreenNumber", 2)
   TextField "HmiScreenItemData" at 80,167 size 640x22; Text 'Plan'
   Button "Back" at 1,1 size 159x47; TextOff 'Back'
      on Release: ActivateScreen("Home", 0)
   Button "HmiScreenItemData_1" at 36,95 size 159x47; TextOff 'Unit1'; PictureOff "Navigates to Unit1 for TP900 Comfort 14.0.1.0"; PictureOn "Navigates to Unit1 for TP900 Comfort 14.0.1.0"
      on Release: ActivateScreen("Unit1", 0)
   Button "HmiScreenItemData_2" at 36,154 size 159x47; TextOff 'Unit2'; PictureOff "Navigates to Unit2 for TP900 Comfort 14.0.1.0"; PictureOn "Navigates to Unit2 for TP900 Comfort 14.0.1.0"
      on Release: ActivateScreen("Unit2", 0)
   Button "HmiScreenItemData_3" at 36,213 size 159x47; TextOff 'Unit3'; PictureOff "Navigates to Unit3 for TP900 Comfort 14.0.1.0"; PictureOn "Navigates to Unit3 for TP900 Comfort 14.0.1.0"
      on Release: ActivateScreen("Unit3", 0)

screen "Unit1" 800x420, template "Template_1"
   on GenerateScreen: SetTag("Tag_ScreenNumber", 3)
   Button "Back" at 1,1 size 159x47; TextOff 'Back'
      on Release: ActivateScreen("Plan", 0)
   Circle "Circle_1" at 23,89 size 23x23
      Appearance <- "SW"
   TextField "Text field_1" at 28,121 size 14x20; Text '0'
   Circle "Circle_2" at 55,89 size 23x23
      Appearance <- "SW"
   TextField "Text field_2" at 60,121 size 14x20; Text '1'
   Circle "Circle_3" at 87,89 size 23x23
      Appearance <- "SW"
   TextField "Text field_3" at 92,121 size 14x20; Text '2'
   Circle "Circle_4" at 119,89 size 23x23
      Appearance <- "SW"
   TextField "Text field_4" at 124,121 size 14x20; Text '3'
   Circle "Circle_5" at 151,89 size 23x23
      Appearance <- "SW"
   TextField "Text field_5" at 156,121 size 14x20; Text '4'
   Circle "Circle_6" at 183,89 size 23x23
      Appearance <- "SW"
   TextField "Text field_6" at 188,121 size 14x20; Text '5'
   Circle "Circle_7" at 215,89 size 23x23
      Appearance <- "SW"
   TextField "Text field_7" at 220,121 size 14x20; Text '6'
   Circle "Circle_8" at 247,89 size 23x23
      Appearance <- "SW"
   TextField "Text field_8" at 252,121 size 14x20; Text '7'
   Circle "Circle_9" at 279,89 size 23x23
      Appearance <- "SW"
   TextField "Text field_9" at 284,121 size 14x20; Text '8'
   Circle "Circle_10" at 311,89 size 23x23
      Appearance <- "SW"
   TextField "Text field_10" at 316,121 size 14x20; Text '9'
   Circle "Circle_11" at 343,89 size 23x23
      Appearance <- "SW"
   TextField "Text field_11" at 343,121 size 23x20; Text '10'
   Circle "Circle_12" at 375,89 size 23x23
      Appearance <- "SW"
   TextField "Text field_12" at 375,121 size 23x20; Text '11'
   Circle "Circle_13" at 407,89 size 23x23
      Appearance <- "SW"
   TextField "Text field_13" at 407,121 size 23x20; Text '12'
   Circle "Circle_14" at 439,89 size 23x23
      Appearance <- "SW"
   TextField "Text field_14" at 439,121 size 23x20; Text '13'
   Circle "Circle_15" at 471,89 size 23x23
      Appearance <- "SW"
   TextField "Text field_15" at 471,121 size 23x20; Text '14'
   Circle "Circle_16" at 503,89 size 23x23
      Appearance <- "SW"
   TextField "Text field_16" at 503,121 size 23x20; Text '15'

screen "Unit2" 800x420, template "Template_1"
   on GenerateScreen: SetTag("Tag_ScreenNumber", 4)
   TextField "HmiScreenItemData" at 80,167 size 640x22; Text 'Unit2'
   Button "Back" at 1,1 size 159x47; TextOff 'Back'
      on Release: ActivateScreen("Plan", 0)

screen "Unit3" 800x420, template "Template_1"
   on GenerateScreen: SetTag("Tag_ScreenNumber", 5)
   TextField "HmiScreenItemData" at 80,167 size 640x22; Text 'Unit3'
   Button "Back" at 1,1 size 159x47; TextOff 'Back'
      on Release: ActivateScreen("Plan", 0)

screen "Param" 800x420, template "Template_1"
   on GenerateScreen: SetTag("Tag_ScreenNumber", 6)
   TextField "HmiScreenItemData" at 80,167 size 640x22; Text 'Param'
   Button "Back" at 1,1 size 159x47; TextOff 'Back'
      on Release: ActivateScreen("Home", 0)
   Button "HmiScreenItemData_1" at 36,95 size 159x47; TextOff 'ParamDI'; PictureOff "Navigates to ParamDI for TP900 Comfort 14.0.1.0"; PictureOn "Navigates to ParamDI for TP900 Comfort 14.0.1.0"
      on Release: ActivateScreen("ParamDI", 0)
   Button "HmiScreenItemData_2" at 36,154 size 159x47; TextOff 'ParamAI'; PictureOff "Navigates to ParamAI for TP900 Comfort 14.0.1.0"; PictureOn "Navigates to ParamAI for TP900 Comfort 14.0.1.0"
      on Release: ActivateScreen("ParamAI", 0)
   Button "HmiScreenItemData_3" at 36,213 size 159x47; TextOff 'ParamAO'; PictureOff "Navigates to ParamAO for TP900 Comfort 14.0.1.0"; PictureOn "Navigates to ParamAO for TP900 Comfort 14.0.1.0"
      on Release: ActivateScreen("ParamAO", 0)
   Button "HmiScreenItemData_4" at 36,272 size 159x47; TextOff 'PAramDO'; PictureOff "Navigates to PAramDO for TP900 Comfort 14.0.1.0"; PictureOn "Navigates to PAramDO for TP900 Comfort 14.0.1.0"
      on Release: ActivateScreen("PAramDO", 0)

screen "ParamDI" 800x420, template "Template_1"
   on GenerateScreen: SetTag("Tag_ScreenNumber", 7)
   TextField "HmiScreenItemData" at 80,167 size 640x22; Text 'ParamDI'
   Button "Back" at 1,1 size 159x47; TextOff 'Back'
      on Release: ActivateScreen("Param", 0)

screen "ParamAI" 800x420, template "Template_1"
   on GenerateScreen: SetTag("Tag_ScreenNumber", 8)
   TextField "HmiScreenItemData" at 80,167 size 640x22; Text 'ParamAI'
   Button "Back" at 1,1 size 159x47; TextOff 'Back'
      on Release: ActivateScreen("Param", 0)

screen "ParamAO" 800x420, template "Template_1"
   on GenerateScreen: SetTag("Tag_ScreenNumber", 9)
   TextField "HmiScreenItemData" at 80,167 size 640x22; Text 'ParamAO'
   Button "Back" at 1,1 size 159x47; TextOff 'Back'
      on Release: ActivateScreen("Param", 0)

screen "PAramDO" 800x420, template "Template_1"
   on GenerateScreen: SetTag("Tag_ScreenNumber", 10)
   TextField "HmiScreenItemData" at 80,167 size 640x22; Text 'PAramDO'
   Button "Back" at 1,1 size 159x47; TextOff 'Back'
      on Release: ActivateScreen("Param", 0)

screen "Recipe" 800x420, template "Template_1"
   on GenerateScreen: SetTag("Tag_ScreenNumber", 11)
   TextField "HmiScreenItemData" at 80,167 size 640x22; Text 'Recipe'
   Button "Back" at 1,1 size 159x47; TextOff 'Back'
      on Release: ActivateScreen("Home", 0)
   Button "HmiScreenItemData_1" at 36,95 size 159x47; TextOff 'R1'; PictureOff "Navigates to R1 for TP900 Comfort 14.0.1.0"; PictureOn "Navigates to R1 for TP900 Comfort 14.0.1.0"
      on Release: ActivateScreen("R1", 0)
   Button "HmiScreenItemData_2" at 36,154 size 159x47; TextOff 'R2'; PictureOff "Navigates to R2 for TP900 Comfort 14.0.1.0"; PictureOn "Navigates to R2 for TP900 Comfort 14.0.1.0"
      on Release: ActivateScreen("R2", 0)

screen "R1" 800x420, template "Template_1"
   on GenerateScreen: SetTag("Tag_ScreenNumber", 12)
   TextField "HmiScreenItemData" at 80,167 size 640x22; Text 'R1'
   Button "Back" at 1,1 size 159x47; TextOff 'Back'
      on Release: ActivateScreen("Recipe", 0)

screen "R2" 800x420, template "Template_1"
   on GenerateScreen: SetTag("Tag_ScreenNumber", 13)
   TextField "HmiScreenItemData" at 80,167 size 640x22; Text 'R2'
   Button "Back" at 1,1 size 159x47; TextOff 'Back'
      on Release: ActivateScreen("Recipe", 0)

screen "Trend" 800x420, template "Template_1"
   on GenerateScreen: SetTag("Tag_ScreenNumber", 14)
   TextField "HmiScreenItemData" at 80,167 size 640x22; Text 'Trend'
   Button "Back" at 1,1 size 159x47; TextOff 'Back'
      on Release: ActivateScreen("Home", 0)
   Button "HmiScreenItemData_1" at 36,95 size 159x47; TextOff 'Trend1'; PictureOff "Navigates to Trend1 for TP900 Comfort 14.0.1.0"; PictureOn "Navigates to Trend1 for TP900 Comfort 14.0.1.0"
      on Release: ActivateScreen("Trend1", 0)
   Button "HmiScreenItemData_2" at 36,154 size 159x47; TextOff 'Trend2'; PictureOff "Navigates to Trend2 for TP900 Comfort 14.0.1.0"; PictureOn "Navigates to Trend2 for TP900 Comfort 14.0.1.0"
      on Release: ActivateScreen("Trend2", 0)
   Button "HmiScreenItemData_3" at 36,213 size 159x47; TextOff 'Trend3'; PictureOff "Navigates to Trend3 for TP900 Comfort 14.0.1.0"; PictureOn "Navigates to Trend3 for TP900 Comfort 14.0.1.0"
      on Release: ActivateScreen("Trend3", 0)

screen "Trend1" 800x420, template "Template_1"
   on GenerateScreen: SetTag("Tag_ScreenNumber", 15)
   TextField "HmiScreenItemData" at 80,167 size 640x22; Text 'Trend1'
   Button "Back" at 1,1 size 159x47; TextOff 'Back'
      on Release: ActivateScreen("Trend", 0)

screen "Trend2" 800x420, template "Template_1"
   on GenerateScreen: SetTag("Tag_ScreenNumber", 16)
   TextField "HmiScreenItemData" at 80,167 size 640x22; Text 'Trend2'
   Button "Back" at 1,1 size 159x47; TextOff 'Back'
      on Release: ActivateScreen("Trend", 0)

screen "Trend3" 800x420, template "Template_1"
   on GenerateScreen: SetTag("Tag_ScreenNumber", 17)
   TextField "HmiScreenItemData" at 80,167 size 640x22; Text 'Trend3'
   Button "Back" at 1,1 size 159x47; TextOff 'Back'
      on Release: ActivateScreen("Trend", 0)

screen "System screens" 800x420, template "Template_1"
   on GenerateScreen: SetTag("Tag_ScreenNumber", 18)
   Button "Back" at 1,1 size 159x47; TextOff 'Back'
      on Release: ActivateScreen("Home", 0)
   Button "HmiScreenItemData" at 36,95 size 159x47; TextOff 'SIMATIC PLC watch table'; PictureOff "Navigates to SIMATIC PLC watch table for TP900 Comfort 14.0.1.0"; PictureOn "Navigates to SIMATIC PLC watch table for TP900 Comfort 14.0.1.0"
      on Release: ActivateScreen("SIMATIC PLC watch table", 0)
   Button "HmiScreenItemData_1" at 36,154 size 159x47; TextOff 'Project information'; PictureOff "Navigates to Project information for TP900 Comfort 14.0.1.0"; PictureOn "Navigates to Project information for TP900 Comfort 14.0.1.0"
      on Release: ActivateScreen("Project information", 0)
   Button "HmiScreenItemData_2" at 36,213 size 159x47; TextOff 'System settings'; PictureOff "Navigates to System settings for TP900 Comfort 14.0.1.0"; PictureOn "Navigates to System settings for TP900 Comfort 14.0.1.0"
      on Release: ActivateScreen("System settings", 0)
   Button "HmiScreenItemData_3" at 36,272 size 159x47; TextOff 'User administration'; PictureOff "Navigates to User administration for TP900 Comfort 14.0.1.0"; PictureOn "Navigates to User administration for TP900 Comfort 14.0.1.0"
      on Release: ActivateScreen("User administration", 0)
   Button "HmiScreenItemData_4" at 207,95 size 159x47; TextOff 'System information'; PictureOff "Navigates to System information for TP900 Comfort 14.0.1.0"; PictureOn "Navigates to System information for TP900 Comfort 14.0.1.0"
      on Release: ActivateScreen("System information", 0)
   Button "HmiScreenItemData_5" at 207,154 size 159x47; TextOff 'Different jobs'; PictureOff "Navigates to Different jobs for TP900 Comfort 14.0.1.0"; PictureOn "Navigates to Different jobs for TP900 Comfort 14.0.1.0"
      on Release: ActivateScreen("Different jobs", 0)

screen "SIMATIC PLC watch table" 800x420, template "Template_1"
   on GenerateScreen: SetTag("Tag_ScreenNumber", 19)
   StatusForce "HmiScreenItemData" at 1,49 size 796x304; ToolTipText 'Text'
   Button "Back" at 1,1 size 159x47; TextOff 'Back'
      on Release: ActivateScreen("System screens", 0)

screen "Project information" 800x420, template "Template_1"
   on GenerateScreen: SetTag("Tag_ScreenNumber", 20)
   TextField "HmiScreenItemData" at 35,51 size 171x28; Text 'Project name:'
   TextField "HmiScreenItemData_1" at 241,51 size 524x28; Text 'SVO_Lib'
   TextField "HmiScreenItemData_2" at 35,81 size 171x28; Text 'Created on:'
   TextField "HmiScreenItemData_3" at 241,81 size 524x28; Text '1/19/2018 9:31:08 AM'
   TextField "HmiScreenItemData_4" at 35,111 size 171x28; Text 'Author:'
   TextField "HmiScreenItemData_5" at 241,111 size 524x28; Text 'SlavaSVO'
   TextField "HmiScreenItemData_6" at 35,141 size 171x28; Text 'Description:'
   TextField "HmiScreenItemData_7" at 241,141 size 524x28; Text '(not configured)'
   Button "Back" at 1,1 size 159x47; TextOff 'Back'
      on Release: ActivateScreen("System screens", 0)

screen "System settings" 800x420, template "Template_1"
   on GenerateScreen: SetTag("Tag_ScreenNumber", 21)
   Button "Calibrate screen" at 36,95 size 159x47; TextOff 'Calibrate screen'
      on Release: function_bc3e350c()
   Button "Clean screen" at 36,154 size 159x47; TextOff 'Clean screen'
      on Release: function_be740847(30)
   Button "Back" at 1,1 size 159x47; TextOff 'Back'
      on Release: ActivateScreen("System screens", 0)

screen "User administration" 800x420, template "Template_1"
   on GenerateScreen: SetTag("Tag_ScreenNumber", 22)
   UserView "HmiScreenItemData" at 1,49 size 796x304
   Button "Back" at 1,1 size 159x47; TextOff 'Back'
      on Release: ActivateScreen("System screens", 0)

screen "System information" 800x420, template "Template_1"
   on GenerateScreen: SetTag("Tag_ScreenNumber", 23)
   TextField "HmiScreenItemData" at 35,51 size 171x28; Text 'HMI device type:'
   TextField "HmiScreenItemData_1" at 241,51 size 524x28; Text 'TP900 Comfort 14.0.1.0'
   TextField "HmiScreenItemData_2" at 35,81 size 171x28; Text 'Version:'
   TextField "HmiScreenItemData_3" at 35,111 size 171x28; Text 'Connection:'
   TextField "HmiScreenItemData_4" at 241,111 size 524x28; Text 'ETHERNET'
   TextField "HmiScreenItemData_5" at 35,141 size 171x28; Text 'PLC:'
   TextField "HmiScreenItemData_6" at 241,141 size 524x28; Text 'SIMATIC S7 300/400'
   Button "Display version" at 241,81 size 524x28; TextOff 'Display version'
      on Release: function_febcb963(-1)
   Button "Back" at 1,1 size 159x47; TextOff 'Back'
      on Release: ActivateScreen("System screens", 0)

screen "Different jobs" 800x420, template "Template_1"
   on GenerateScreen: SetTag("Tag_ScreenNumber", 24)
   Button "Online" at 36,95 size 159x47; TextOff 'Online'
      on Release: function_bb44b551(0)
   Button "Offline" at 36,154 size 159x47; TextOff 'Offline'
      on Release: function_bb44b551(1)
   Button "Transfer" at 36,213 size 159x47; TextOff 'Transfer'
      on Release: function_bb44b551(2)
   Button "Toggle language" at 36,272 size 159x47; TextOff 'Toggle language'
      on Release: function_fb9197e8(-1)
   Button "Control Panel" at 207,95 size 159x47; TextOff 'Control Panel'
      on Release: function_f34a74f3()
   Button "Stop Runtime" at 207,154 size 159x47; TextOff 'Stop Runtime'
      on Release: StopRuntime(0)
   Button "Back" at 1,1 size 159x47; TextOff 'Back'
      on Release: ActivateScreen("System screens", 0)
*)